FUNCTION_BLOCK FB_BA_MeasuredValueCardinal EXTENDS FB_BA_View
VAR_INPUT
	fVal_N					: REAL;
	fVal_S					: REAL;
	fVal_E					: REAL;
	fVal_W					: REAL;
END_VAR
VAR_INPUT CONSTANT
	MV_N					: FB_BA_AI;		
	MV_S					: FB_BA_AI;	
	MV_E					: FB_BA_AI;		
	MV_W					: FB_BA_AI;			
END_VAR
VAR_OUTPUT
	fPresentValueN			: REAL;
	fPresentValueS			: REAL;
	fPresentValueE			: REAL;
	fPresentValueW			: REAL;
END_VAR
VAR
END_VAR

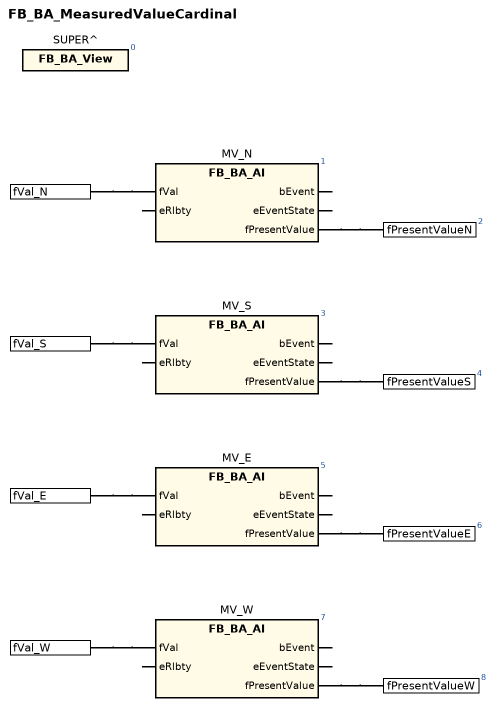
SUPER^(); // FB_BA_View
MV_N(fVal := fVal_N); // FB_BA_AI
fPresentValueN := MV_N.fPresentValue;
MV_S(fVal := fVal_S); // FB_BA_AI
fPresentValueS := MV_S.fPresentValue;
MV_E(fVal := fVal_E); // FB_BA_AI
fPresentValueE := MV_E.fPresentValue;
MV_W(fVal := fVal_W); // FB_BA_AI
fPresentValueW := MV_W.fPresentValue;

METHOD FB_init : BOOL
VAR_INPUT
	bInitRetains : BOOL; // if TRUE, the retain variables are initialized (warm start / cold start)
	bInCopyCode : BOOL;  // if TRUE, the instance afterwards gets moved into the copy code (online change)
END_VAR
MV_N.iParent						:= THIS^;		
MV_N.iLabel 						:= LblUniFieldDevice.SensorAnalog_MV_N;
MV_N.sObjectName					:= '{Idx=01}';
MV_N.sDeviceType					:= '';
MV_N.bEnOutOfService				:= FALSE;
MV_N.eUnit							:= E_BA_Unit.eTemperature_DegreesCelsius;
MV_N.fResolution 					:= 0.01;
MV_N.fScaleOffset 					:= 0; 	
MV_N.fCOVIncrement					:= BA2_Param.fDefCOVIncrement;
MV_N.nEventClassID					:= EventClasses.AlarmTechnicalExtended;
MV_N.stTimeDelay.nToNormal			:= BA2_Param.nDefTimeDelay_ToNormal;
MV_N.stTimeDelay.nToAbnormal		:= BA2_Param.nDefTimeDelay_ToAbnormal;
MV_N.stHighLimit.bEnable			:= FALSE;
MV_N.stHighLimit.fValue				:= 0.0;		
MV_N.stLowLimit.bEnable				:= FALSE;
MV_N.stLowLimit.fValue				:= 0.0;
MV_N.fLimitDeadband 				:= BA2_Param.fDefLimitDeadband;
MV_N.bAcknowledgeRm					:= FALSE;	
MV_N.aEventTransitionText[1]		:= Texts.txtExceeded;
MV_N.aEventTransitionText[2]		:= Texts.txtDisturb;
MV_N.aEventTransitionText[3]		:= Texts.txtNormal;
MV_N.bEventDetectionEnable			:= FALSE;
MV_N.eEnPlantLock					:= E_BA_LockPriority.eNoLock;			

MV_S.iParent						:= THIS^;		
MV_S.iLabel 						:= LblUniFieldDevice.SensorAnalog_MV_S;
MV_S.sObjectName					:= '{Idx=01}';
MV_S.sDeviceType					:= '';
MV_S.bEnOutOfService				:= FALSE;
MV_S.eUnit							:= E_BA_Unit.eTemperature_DegreesCelsius;
MV_S.fResolution 					:= 0.01;
MV_S.fScaleOffset 					:= 0; 	
MV_S.fCOVIncrement					:= BA2_Param.fDefCOVIncrement;
MV_S.nEventClassID					:= EventClasses.AlarmTechnicalExtended;
MV_S.stTimeDelay.nToNormal			:= BA2_Param.nDefTimeDelay_ToNormal;
MV_S.stTimeDelay.nToAbnormal		:= BA2_Param.nDefTimeDelay_ToAbnormal;
MV_S.stHighLimit.bEnable			:= FALSE;
MV_S.stHighLimit.fValue				:= 0.0;		
MV_S.stLowLimit.bEnable				:= FALSE;
MV_S.stLowLimit.fValue				:= 0.0;
MV_S.fLimitDeadband 				:= BA2_Param.fDefLimitDeadband;
MV_S.bAcknowledgeRm					:= FALSE;	
MV_S.aEventTransitionText[1]		:= Texts.txtExceeded;
MV_S.aEventTransitionText[2]		:= Texts.txtDisturb;
MV_S.aEventTransitionText[3]		:= Texts.txtNormal;
MV_S.bEventDetectionEnable			:= FALSE;
MV_S.eEnPlantLock					:= E_BA_LockPriority.eNoLock;

MV_E.iParent						:= THIS^;		
MV_E.iLabel 						:= LblUniFieldDevice.SensorAnalog_MV_E;
MV_E.sObjectName					:= '{Idx=01}';
MV_E.sDeviceType					:= '';
MV_E.bEnOutOfService				:= FALSE;
MV_E.eUnit							:= E_BA_Unit.eTemperature_DegreesCelsius;
MV_E.fResolution 					:= 0.01;
MV_E.fScaleOffset 					:= 0; 	
MV_E.fCOVIncrement					:= BA2_Param.fDefCOVIncrement;
MV_E.nEventClassID					:= EventClasses.AlarmTechnicalExtended;
MV_E.stTimeDelay.nToNormal			:= BA2_Param.nDefTimeDelay_ToNormal;
MV_E.stTimeDelay.nToAbnormal		:= BA2_Param.nDefTimeDelay_ToAbnormal;
MV_E.stHighLimit.bEnable			:= FALSE;
MV_E.stHighLimit.fValue				:= 0.0;		
MV_E.stLowLimit.bEnable				:= FALSE;
MV_E.stLowLimit.fValue				:= 0.0;
MV_E.fLimitDeadband 				:= BA2_Param.fDefLimitDeadband;
MV_E.bAcknowledgeRm					:= FALSE;	
MV_E.aEventTransitionText[1]		:= Texts.txtExceeded;
MV_E.aEventTransitionText[2]		:= Texts.txtDisturb;
MV_E.aEventTransitionText[3]		:= Texts.txtNormal;
MV_E.bEventDetectionEnable			:= FALSE;
MV_E.eEnPlantLock					:= E_BA_LockPriority.eNoLock;

MV_W.iParent						:= THIS^;		
MV_W.iLabel 						:= LblUniFieldDevice.SensorAnalog_MV_W;
MV_W.sObjectName					:= '{Idx=01}';
MV_W.sDeviceType					:= '';
MV_W.bEnOutOfService				:= FALSE;
MV_W.eUnit							:= E_BA_Unit.eTemperature_DegreesCelsius;
MV_W.fResolution 					:= 0.01;
MV_W.fScaleOffset 					:= 0; 	
MV_W.fCOVIncrement					:= BA2_Param.fDefCOVIncrement;
MV_W.nEventClassID					:= EventClasses.AlarmTechnicalExtended;
MV_W.stTimeDelay.nToNormal			:= BA2_Param.nDefTimeDelay_ToNormal;
MV_W.stTimeDelay.nToAbnormal		:= BA2_Param.nDefTimeDelay_ToAbnormal;
MV_W.stHighLimit.bEnable			:= FALSE;
MV_W.stHighLimit.fValue				:= 0.0;		
MV_W.stLowLimit.bEnable				:= FALSE;
MV_W.stLowLimit.fValue				:= 0.0;
MV_W.fLimitDeadband 				:= BA2_Param.fDefLimitDeadband;
MV_W.bAcknowledgeRm					:= FALSE;	
MV_W.aEventTransitionText[1]		:= Texts.txtExceeded;
MV_W.aEventTransitionText[2]		:= Texts.txtDisturb;
MV_W.aEventTransitionText[3]		:= Texts.txtNormal;
MV_W.bEventDetectionEnable			:= FALSE;
MV_W.eEnPlantLock					:= E_BA_LockPriority.eNoLock;
END_METHOD

END_FUNCTION_BLOCK

(* stored: Version 1.1.0.1, ProductVersion 3.1.4024.6
   POU FB_BA_MeasuredValueCardinal: Id {3ea16385-8aaa-40ca-82d6-c83eaad72ee1}, SpecialFunc None
   Method FB_init: Id {1b39da57-7d5c-49f7-b602-76b6bfd1cbf4} *)
